FUNCTION_BLOCK pingerfb (* JADE WORKER *)
  (* Standard: 61499-1 *)
  (* Version 1.0, 2014-04-22, Ahmed, Fraunhofer IGD *)
  (* Compiler header: package fb.rt; *)
  (* Compiler Java Sun JDK 1.5.0 *)
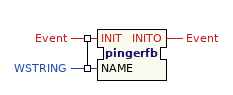
  EVENT_INPUT
    INIT WITH NAME; (* Normal Execution Request *)
  END_EVENT
  EVENT_OUTPUT
    INITO; (* Execution Confirmation *)
  END_EVENT
  VAR_INPUT
    NAME : WSTRING;
  END_VAR
END_FUNCTION_BLOCK
